PROGRAM POU_MAIN_UML_StateChart
VAR
		bStartProcess	:	BOOL	:=	FALSE;
END_VAR

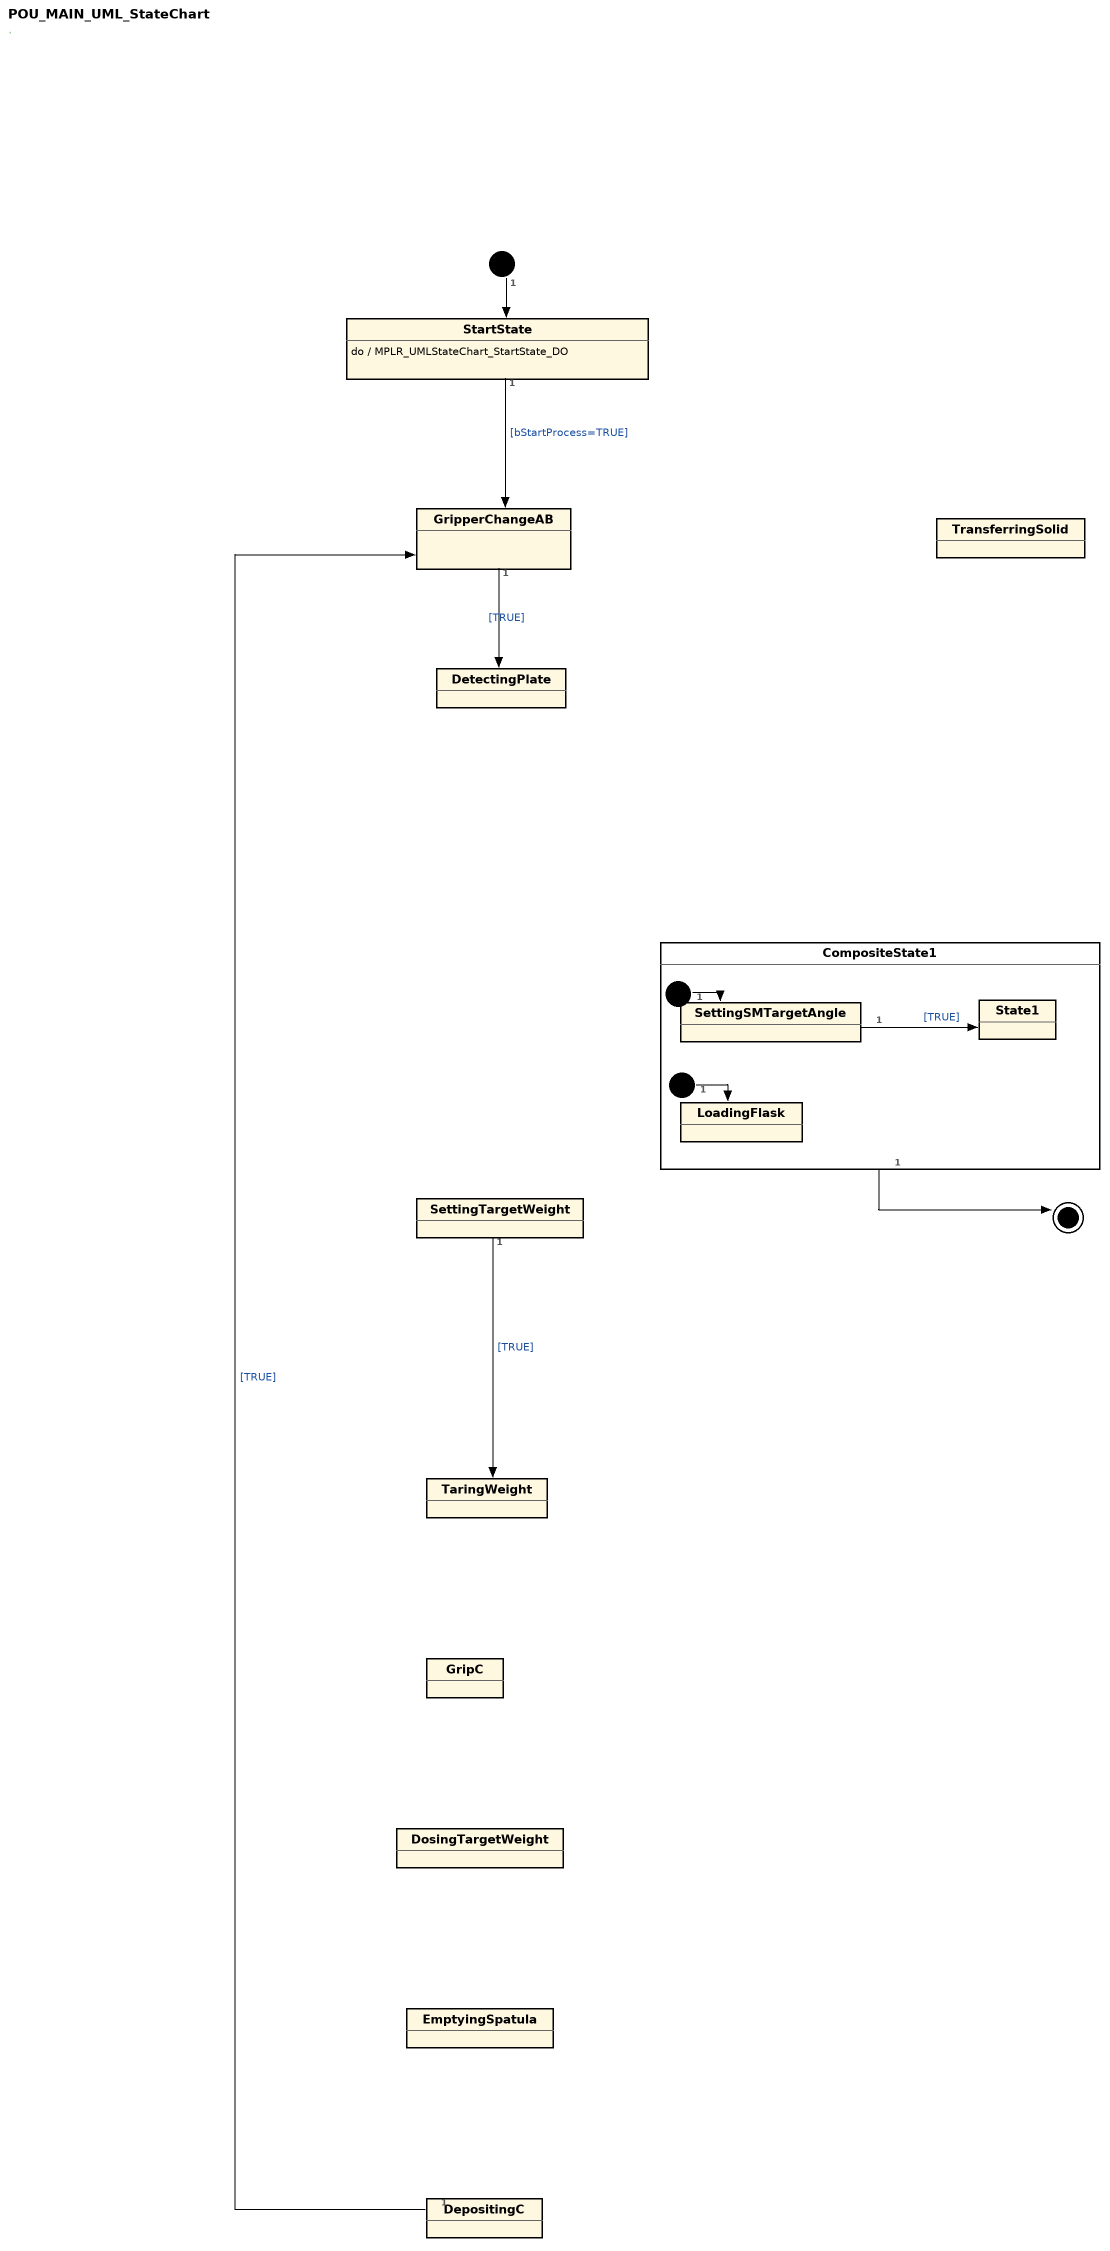
STATECHART POU_MAIN_UML_StateChart  // abortable
    START StartState1
    NOTEELEMENT 
    NOTEELEMENT 
    NOTEELEMENT 
    STATE StartState
        do / MPLR_UMLStateChart_StartState_DO
    STATE GripperChangeAB
    STATE TransferringSolid
    STATE DetectingPlate
    COMPOSITE STATE CompositeState1
        REGION Region1 // priority 1
        START StartState3
        STATE LoadingFlask
        StartState3 -> LoadingFlask  // priority 1, on completion
        REGION Region0 // priority 2
        START StartState2
        STATE SettingSMTargetAngle
        STATE State1
        StartState2 -> SettingSMTargetAngle  // priority 1, on completion
        SettingSMTargetAngle -> State1 [TRUE] // priority 1
    END_STATE
    STATE SettingTargetWeight
    END EndState1
    STATE TaringWeight
    STATE GripC
    STATE DosingTargetWeight
    STATE EmptyingSpatula
    STATE DepositingC
    StartState1 -> StartState  // priority 1, on completion
    StartState -> GripperChangeAB [bStartProcess=TRUE] // priority 1
    GripperChangeAB -> DetectingPlate [TRUE] // priority 1
    CompositeState1 -> EndState1  // priority 1, on completion
    SettingTargetWeight -> TaringWeight [TRUE] // priority 1
    DepositingC -> GripperChangeAB [TRUE] // priority 1
END_STATECHART

END_PROGRAM

(* stored: Version 1.1.0.1
   POU POU_MAIN_UML_StateChart: Id {e2cfee17-0e64-4677-a08f-fafba64656a0}, SpecialFunc None *)
